(* PLC project v0.6.04_CycleSemiAuto.project, CODESYS CODESYS V3.5 SP19 Patch 1 *)
(* stored: creationDateTime 2026-07-23T23:21:28.108376, modificationDateTime 2026-07-23T23:21:28.108376 *)

(* ═══════════════════════════════════════════════════════════════ 🔧 ST_SyncCfg — Configuration de la synchronisation M1/M2 ═══════════════════════════════════════════════════════════════ *)
TYPE ST_SyncCfg : STRUCT
  CfgSyncTolerance_M : REAL := 0.8;  (* 📐 Tolérance max d'écart (m) — Dégradation Palier 1 dès 0.8m *)
  Initialized : BOOL := FALSE;  (* 🚦 flag restauration boot, ex-CfgInitialized renommé pour cohérence avec ST_WinchCfg *)
END_STRUCT;
END_TYPE

(* ═══════════════════════════════════════════════════════════════ 🌉 FB_CfgPersistBridge_SyncCfg — Pont persistance générique pour ST_SyncCfg ─────────────────────────────────────────────────────────────── 🎯 Remplace les blocs manuels restauration/sauvegarde dupliqués à chaque domaine (voir DOC/AUDITS/ConfigPersistence/). Une instance = un couple (struct IHM, struct GVL_PERSISTENT) du MÊME type. Logique : - Hmi.Initialized = FALSE (RETAIN invalidé, ex. changement de layout DUT) → restaure Hmi depuis Persist, marque Initialized, pulse JustRestored 1 scan. - Hmi.Initialized = TRUE → sauvegarde continue Hmi vers Persist (jamais l'inverse). 🔒 Défense en profondeur : jamais d'écriture PERSISTENT avant qu'une restauration réussie n'ait eu lieu (même principe que tous les blocs Cfg du Lot 2). ═══════════════════════════════════════════════════════════════ *)
FUNCTION_BLOCK FB_CfgPersistBridge_SyncCfg
  VAR_OUTPUT
    JustRestored : BOOL;  (* 🔔 TRUE pendant 1 scan le boot où la restauration a eu lieu — *)
  END_VAR
  VAR_IN_OUT
    Hmi : ST_SyncCfg;  (* 🖥️ ex. GVL_IHM.M1M2Sync.Cfg — struct exposé à l'IHM *)
    Persist : ST_SyncCfg;  (* 💾 ex. GVL_PERSISTENT._SyncCfgPersist — mémoire PERSISTENT *)
  END_VAR

            

JustRestored := FALSE;
IF NOT Hmi.Initialized THEN
    Hmi := Persist;
    Hmi.Initialized := TRUE;
    JustRestored := TRUE;
ELSE
    Persist := Hmi;
END_IF;

          
END_FUNCTION_BLOCK
